TYPE ST_InfoDataConnection_1904 :
STRUCT
	usiMapState: USINT;
	usiMapDiag: USINT;
	bySignals: BYTE;
END_STRUCT
END_TYPE

(* stored: Version 1.1.0.1
   DUT ST_InfoDataConnection_1904: Id {2deb761b-1c22-48e4-994d-ada17e1181c7} *)
